(* CoDeSys 2.3 export: TRANSFER_TO_2_10B.EXP *)

(* POU Transfer_To_2_10B, ST *)
FUNCTION Transfer_To_2_10B : REAL
VAR_INPUT
	IN: REAL;				(* input value*)
END_VAR
VAR
	IN_MIN:REAL := 0;			(* minimum input value *)
	IN_MAX:REAL := 1;			(* maximum input value *)
	OUT_MIN:REAL := 0.2;		(* corresponding minimum output value *)
	OUT_MAX:REAL  := 1;		(* corresponding maximum output value *)
	Diff: REAL;
END_VAR
	Diff := IN_MAX-IN_MIN;
	Transfer_To_2_10B := (IN-IN_MIN)/Diff * (OUT_MAX-OUT_MIN) + OUT_MIN;
END_FUNCTION
